FUNCTION_BLOCK SteamLimit (* Basic Function Block Type *)
  (* Standard: 61499-2 *)
  (* Version 0.0, 2011-12-23, 4DIAC-IDE, 4DIAC-Consortium *)
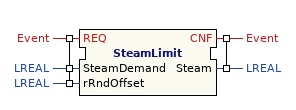
  EVENT_INPUT
    REQ WITH SteamDemand, rRndOffset; (* Normal Execution Request *)
  END_EVENT
  EVENT_OUTPUT
    CNF WITH Steam; (* Execution Confirmation *)
  END_EVENT
  VAR_INPUT
    SteamDemand : LREAL; (* Input event qualifier *)
    rRndOffset : LREAL;
  END_VAR
  VAR_OUTPUT
    Steam : LREAL; (* Output event qualifier *)
  END_VAR
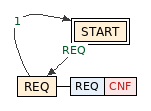
  EC_STATES
    START; (* Initial State *)
    REQ : REQ -> CNF; (* Normal execution *)
  END_STATES
  EC_TRANSITIONS
    START TO REQ := REQ;
    REQ TO START := 1;
  END_TRANSITIONS
  ALGORITHM REQ IN ST: (* Normally executed algorithm *)
IF (SteamDemand+rRndOffset) >=10 THEN
	Steam:=10;
ELSE
	IF  (SteamDemand+rRndOffset) <=0 THEN
		Steam:=0;
	ELSE
		Steam:=SteamDemand+rRndOffset;
	END_IF;
END_IF;
  END_ALGORITHM
END_FUNCTION_BLOCK
